// TIA Portal V18 export
TYPE "UDT_signalColumn"
// stored: IsFailsafeCompliant false
   STRUCT
      O_green { ExternalVisible := 'False'; ExternalWritable := 'False'} : Bool;
      O_yellow { ExternalVisible := 'False'; ExternalWritable := 'False'} : Bool;
      O_red { ExternalVisible := 'False'; ExternalWritable := 'False'} : Bool;
   END_STRUCT;
END_TYPE
